// TwinCAT 3 PLC project PLC1
// ProgramVersion: 3.1.4024.0
// libraries:
//   Tc2_Standard, * (Beckhoff Automation GmbH)
//   Tc2_System, * (Beckhoff Automation GmbH)
//   Tc3_Module, * (Beckhoff Automation GmbH)
// project tree:
//   DUTs/ DUT_IncomingMsgRequest.TcDUT, DUT_MsgToAmsPortHeader.TcDUT, DUT_OutgoingMsgResponse.TcDUT
//   GVLs/ CONST.TcGVL
//   / PlcTask.TcTTO
//   POUs/ MAIN.TcPOU
// real-time tasks:
//   TASK PlcTask: cycle T#10ms, priority 20, ADS port 350
//   TASK EIP_Task: cycle T#1ms, priority 2, ADS port 301
// I/O:
//   DEVICE Device 1 (TC3 EIP Adapter), AmsNetId 5.58.183.60.2.1
//     C6032_TF6280

CONFIGURATION PLC1
    RESOURCE PLC ON TwinCAT3
        TASK PlcTask(INTERVAL := T#10ms, PRIORITY := 20);
        PROGRAM MAIN WITH PlcTask : MAIN;
    END_RESOURCE
END_CONFIGURATION

// ---- DUTs/DUT_IncomingMsgRequest.TcDUT
TYPE
    DUT_IncomingMsgRequest :
    STRUCT
        reqHdr : DUT_MsgToAmsPortHeader;
        reqData : ARRAY[0..991] OF BYTE;
    END_STRUCT
END_TYPE

// ---- DUTs/DUT_MsgToAmsPortHeader.TcDUT
TYPE
    DUT_MsgToAmsPortHeader :
    STRUCT
        nServiceCode : UDINT;
        nClassId : UDINT;
        nInstanceId : UDINT;
        nAttributeId : UDINT;
        nReservedId : UDINT;
        nGeneralStatus : UDINT;
        nAdditionalStatus : UDINT;
        nDataLen : UDINT;
    END_STRUCT
END_TYPE

// ---- DUTs/DUT_OutgoingMsgResponse.TcDUT
TYPE
    DUT_OutgoingMsgResponse :
    STRUCT
        resHdr : DUT_MsgToAmsPortHeader;
        resData : ARRAY[0..991] OF BYTE;
    END_STRUCT
END_TYPE

// ---- GVLs/CONST.TcGVL
{attribute 'qualified_only'}
VAR_GLOBAL CONSTANT
    //Service Codes
    CN_SC_REPLY_MASK : BYTE := 16#80;
    CN_SC_GET_ATTR_SINGLE : BYTE := 16#0E;
    CN_SC_SET_ATTR_SINGLE : BYTE := 16#10;

    //MPath Segment Types
    CN_LOGICAL_SEGMENT : BYTE := 16#20;

    CN_LOGICAL_SEG_CLASS : BYTE := 16#00;
    CN_LOGICAL_SEG_INSTANCE : BYTE := 16#04;
    CN_LOGICAL_SEG_STRUCT : BYTE := 16#08;
    CN_LOGICAL_SEG_ATTRIBUTE : BYTE := 16#10;

    CN_LOGICAL_SEG_8_BIT : BYTE := 16#00;
    CN_LOGICAL_SEG_16_BIT : BYTE := 16#01;
    CN_LOGICAL_SEG_32_BIT : BYTE := 16#02;

    CN_IOI_SEG_CLASS_8 : BYTE := CN_LOGICAL_SEGMENT OR CN_LOGICAL_SEG_CLASS OR CN_LOGICAL_SEG_8_BIT;
    CN_IOI_SEG_CLASS_16 : BYTE := CN_LOGICAL_SEGMENT OR CN_LOGICAL_SEG_CLASS OR CN_LOGICAL_SEG_16_BIT;
    CN_IOI_SEG_CLASS_32 : BYTE := CN_LOGICAL_SEGMENT OR CN_LOGICAL_SEG_CLASS OR CN_LOGICAL_SEG_32_BIT;

    CN_IOI_SEG_INSTANCE_8 : BYTE := CN_LOGICAL_SEGMENT OR CN_LOGICAL_SEG_INSTANCE OR CN_LOGICAL_SEG_8_BIT;
    CN_IOI_SEG_INSTANCE_16 : BYTE := CN_LOGICAL_SEGMENT OR CN_LOGICAL_SEG_INSTANCE OR CN_LOGICAL_SEG_16_BIT;
    CN_IOI_SEG_INSTANCE_32 : BYTE := CN_LOGICAL_SEGMENT OR CN_LOGICAL_SEG_INSTANCE OR CN_LOGICAL_SEG_32_BIT;

    CN_IOI_SEG_MEMBER_8 : BYTE := CN_LOGICAL_SEGMENT OR CN_LOGICAL_SEG_STRUCT OR CN_LOGICAL_SEG_8_BIT;
    CN_IOI_SEG_MEMBER_16 : BYTE := CN_LOGICAL_SEGMENT OR CN_LOGICAL_SEG_STRUCT OR CN_LOGICAL_SEG_16_BIT;
    CN_IOI_SEG_MEMBER_32 : BYTE := CN_LOGICAL_SEGMENT OR CN_LOGICAL_SEG_STRUCT OR CN_LOGICAL_SEG_32_BIT;

    CN_IOI_SEG_ATTRIBUTE_8 : BYTE := CN_LOGICAL_SEGMENT OR CN_LOGICAL_SEG_ATTRIBUTE OR CN_LOGICAL_SEG_8_BIT;
    CN_IOI_SEG_ATTRIBUTE_16 : BYTE := CN_LOGICAL_SEGMENT OR CN_LOGICAL_SEG_ATTRIBUTE OR CN_LOGICAL_SEG_16_BIT;
    CN_IOI_SEG_ATTRIBUTE_32 : BYTE := CN_LOGICAL_SEGMENT OR CN_LOGICAL_SEG_ATTRIBUTE OR CN_LOGICAL_SEG_32_BIT;

    //General Status Codes
    CN_GRC_SUCCESS : BYTE := 16#00; // We done good...               */
    CN_GRC_CONNECTION_FAILURE : BYTE := 16#01; // A connection related service failed along the connection path.             */
    CN_GRC_NO_RESOURCE : BYTE := 16#02; // Resource(S) unavailable       */
    CN_GRC_BAD_DATA : BYTE := 16#03; // Obj specific data bad         */
    CN_GRC_BAD_IOI : BYTE := 16#04; // IOI hosed                     */
    CN_GRC_BAD_CLASS_INSTANCE : BYTE := 16#05; // Class/instance unknown        */
    CN_GRC_PARTIAL_DATA : BYTE := 16#06; // NOT all expected data sent    */
    CN_GRC_CONN_LOST : BYTE := 16#07; // Messaging connection lost     */
    CN_GRC_BAD_SERVICE : BYTE := 16#08; // Unimplimented service code    */
    CN_GRC_BAD_ATTR_DATA : BYTE := 16#09; // Bad attribute data value      */
    CN_GRC_ATTR_LIST_ERROR : BYTE := 16#0A; // Get/set attr list failed      */
    CN_GRC_ALREADY_IN_MODE : BYTE := 16#0B; // Obj already in requested mode */
    CN_GRC_BAD_OBJ_MODE : BYTE := 16#0C; // Obj NOT in proper mode        */
    CN_GRC_OBJ_ALREADY_EXISTS : BYTE := 16#0D; // Object already created        */
    CN_GRC_ATTR_NOT_SETTABLE : BYTE := 16#0E; // Set OF get only attr tried    */
    CN_GRC_PERMISSION_DENIED : BYTE := 16#0F; // Insufficient access permission*/
    CN_GRC_SET_ATTR_WRONG_STATE : BYTE := 16#10; // Set attribute NOT allowed     */
    CN_GRC_RESPONSE_TOO_LARGE : BYTE := 16#11; // Response packet too large     */
    CN_GRC_CONFIG_TOO_SMALL : BYTE := 16#13; // Goldilocks complaint #1       */
    CN_GRC_UNDEFINED_ATTR : BYTE := 16#14; // Attribute is undefined        */
    CN_GRC_CONFIG_TOO_BIG : BYTE := 16#15; // Goldilocks complaint #2       */
    CN_GRC_OBJ_NOT_EXISTING : BYTE := 16#16; // The object specified does NOT exist in the divce*/
    CN_GRC_VENDOR_SPECIFIC_ERR : BYTE := 16#1F; //
    CN_GRC_INVALID_PARAMETER : BYTE := 16#20; //
    CN_GRC_BAD_KEY_IN_IOI : BYTE := 16#25; // Electronic key in IOI failed  */
    CN_GRC_BAD_IOI_SIZE : BYTE := 16#26; // Invalid IOI size              */

    //Additional Status Codes
    CN_ORC_NO_BUFFER : WORD := 16#0301; // No buffer memory available    */
    CN_ORC_BAD_SEGMENT : WORD := 16#0315; // Invalid segment in path       */
END_VAR

// ---- POUs/MAIN.TcPOU
PROGRAM MAIN
VAR
    i : INT;
    IdxGroup : UDINT;
    IdxOffset : UDINT;
    fbAdsRdWrInd : ADSRDWRTIND;
    fbAdsRdWrRes : ADSRDWRTRES;
    request : DUT_IncomingMsgRequest;
    response : DUT_OutgoingMsgResponse;
    nResponseLen : UINT;
    nAdsResult : UDINT := 0;
    nAdsResponsesSent : UDINT;
    Attributes : ARRAY[1..4] OF STRING := ['TestReadOnlyAttribute1', 'TestReadOnlyAttribute2', 'TestReadOnlyAttribute3', '1'];
    fbADSRDWRTINDEX : ADSRDWRTINDEX;
END_VAR

CASE i OF

    0: fbADSRDWRTINDEX(CLEAR := FALSE,
            MINIDXGRP := 16#84000000,
            VALID =>,
            NETID =>,
            PORT =>,
            INVOKEID =>,
            IDXGRP =>,
            IDXOFFS =>,
            RDLENGTH =>,
            WRTLENGTH =>,
            DATAADDR =>);

        IF fbADSRDWRTINDEX.VALID THEN
            IdxGroup := fbADSRDWRTINDEX.IDXGRP;
            IdxOffset := fbADSRDWRTINDEX.IDXOFFS;
            nResponseLen := 0;
            MEMSET(ADR(request), 0, SIZEOF(request));
            MEMSET(ADR(response), 0, SIZEOF(response));

            IF IdxGroup = 16#848180E9 THEN
                IF fbADSRDWRTINDEX.WRTLENGTH >= SIZEOF(request.reqHdr) THEN
                    MEMCPY(ADR(request.reqHdr), fbADSRDWRTINDEX.DATAADDR, SIZEOF(request.reqHdr));
                END_IF

                IF fbADSRDWRTINDEX.WRTLENGTH > SIZEOF(request.reqHdr) THEN
                    MEMCPY(ADR(request.reqData),
                        fbADSRDWRTINDEX.DATAADDR + SIZEOF(request.reqHdr),
                        fbADSRDWRTINDEX.WRTLENGTH - SIZEOF(request.reqHdr));
                END_IF

                i := 10;
            ELSE
                i := 20;
            END_IF
        END_IF

    10: //new Ind from EthIp-Drv received
        response.resHdr.nServiceCode := request.reqHdr.nServiceCode OR CONST.CN_SC_REPLY_MASK;
        response.resHdr.nGeneralStatus := 0;
        response.resHdr.nAdditionalStatus := 0;
        response.resHdr.nDataLen := 0;

        IF request.reqHdr.nServiceCode = CONST.CN_SC_GET_ATTR_SINGLE OR request.reqHdr.nServiceCode = CONST.CN_SC_SET_ATTR_SINGLE THEN
            i := 11;
        ELSE
            response.resHdr.nGeneralStatus := CONST.CN_GRC_BAD_SERVICE;
            nResponseLen := SIZEOF(response.resHdr);
            i := 20;
        END_IF

    11: CASE request.reqHdr.nClassId OF
            16#1000: //erlaubte Beispiel Class 0x10000
                CASE request.reqHdr.nInstanceId OF
                    16#1: //erlaubte Beispiel Instance 0x1
                        CASE request.reqHdr.nAttributeId OF //Attributes 1-4 erlaubt; only attr 4 is settable 
                            1, 2, 3: IF request.reqHdr.nServiceCode = CONST.CN_SC_SET_ATTR_SINGLE THEN
                                    response.resHdr.nGeneralStatus := CONST.CN_GRC_ATTR_NOT_SETTABLE;
                                    nResponseLen := SIZEOF(response.resHdr);
                                    i := 20;
                                ELSE
                                    i := 12;
                                END_IF
                            4: IF request.reqHdr.nServiceCode = CONST.CN_SC_SET_ATTR_SINGLE THEN
                                    i := 14;
                                ELSE
                                    i := 12;
                                END_IF
                        ELSE
                            response.resHdr.nGeneralStatus := CONST.CN_GRC_UNDEFINED_ATTR;
                            nResponseLen := SIZEOF(response.resHdr);
                            i := 20;
                        END_CASE
                ELSE
                    response.resHdr.nGeneralStatus := CONST.CN_GRC_BAD_CLASS_INSTANCE;
                    nResponseLen := SIZEOF(response.resHdr);
                    i := 20;
                END_CASE
        ELSE
            response.resHdr.nGeneralStatus := CONST.CN_GRC_BAD_CLASS_INSTANCE;
            nResponseLen := SIZEOF(response.resHdr);
            i := 20;
        END_CASE

    12: //GetAttribute
        response.resHdr.nGeneralStatus := CONST.CN_GRC_SUCCESS;
        MEMCPY(ADR(response.resData), ADR(Attributes[request.reqHdr.nAttributeId]), SIZEOF(Attributes[request.reqHdr.nAttributeId]));
        response.resHdr.nDataLen := INT_TO_UINT(LEN(Attributes[request.reqHdr.nAttributeId]));
        nResponseLen := UDINT_TO_UINT(response.resHdr.nDataLen) + SIZEOF(response.resHdr);
        i := 20;

    14: //SetAttribute	
        response.resHdr.nGeneralStatus := CONST.CN_GRC_SUCCESS;

        IF request.reqHdr.nDataLen <= SIZEOF(STRING) - 1 THEN
            MEMCPY(ADR(Attributes[request.reqHdr.nAttributeId]), ADR(request.reqData), request.reqHdr.nDataLen);
        ELSE
            response.resHdr.nGeneralStatus := CONST.CN_GRC_BAD_DATA; //zuviel Schreibdaten
        END_IF

        nResponseLen := SIZEOF(response.resHdr);
        i := 20;

    20: fbAdsRdWrRes(NETID := fbADSRDWRTINDEX.NETID,
            PORT := fbADSRDWRTINDEX.PORT,
            INVOKEID := fbADSRDWRTINDEX.INVOKEID,
            RESULT := nAdsResult,
            LEN := nResponseLen,
            DATAADDR := ADR(Response),
            RESPOND := TRUE);

        i := 21;
        nAdsResponsesSent := nAdsResponsesSent + 1;
        fbADSRDWRTINDEX(CLEAR := TRUE);
    21: i := 0;
        fbAdsRdWrRes(RESPOND := FALSE);
END_CASE

END_PROGRAM
